(* PLC project Rasi_feeds_batching.project, Automation Builder 2.7 - Basic Automation Builder 2.7 *)
(* stored: creationDateTime 2026-08-31T23:45:00 *)

TYPE Modbus_Poll_Request : STRUCT
  Slave_ID : BYTE;
  Func_Code : BYTE;
  Start_Reg : WORD;
  Num_Regs : WORD;
  Raw_Data : ARRAY[1..4] OF WORD;
  Done : BOOL;
  Error : BOOL;
  Error_Code : WORD;
END_STRUCT;
END_TYPE
